// Block: MES_Send_Buffer_Msg_Topic3XX

DATA_BLOCK MES_Send_Buffer_Msg_Topic3XX
VERSION : 0.1
   NON_RETAIN
   VAR
      lastId : DInt;
      Counter : DInt;
      msg : Array[1..MES_MSG_ITEMS] of MES_Msg;
   END_VAR

BEGIN
   // No initialization required
END_DATA_BLOCK
